Staubli VAL3: printToShow.pgx

program printToShow()
  local num l_nSize
  local string l_sMessage
  local num l_nScrool
  local bool l_bInside
begin
  //
  //  Print the instruction and the function KEY STEP
  //
  call use:typeLen(0,12,""+cycleStatus:sToShow,40)
  //
  // refresh the scroll bar in simulation
  //
  if cycleStatus:bSimulation
    nMoveId=getMoveId()
  endIf
  if nMoveId>=1
    call trajType:getSizeItem(false,l_nSize)
    // normal point
    call use:type(0,11,toString("2",nPoint)+" ")
    call use:type(37,11,toString("2",nPoint+1)+" ")
  else
    // start Point
    call use:type(0,11,toString("2",nPoint)+" ")
    call use:type(37,11,toString("2",nPoint+1)+" ")
  endIf
  // print the scroll
  call isAtPoint(nPoint,l_bInside)
  if l_bInside
    l_nScrool=100
  else
    l_nScrool=abs(roundDown(nMoveId)-nMoveId)*100
  endIf
  call use:scroll(3,11,32,l_nScrool)
  call language:message(l_sMessage,124)
end
